{attribute 'qualified_only'}
VAR_GLOBAL
	bGetUp : BOOL := TRUE;
	bReady : BOOL;
END_VAR

(* stored: Version 1.1.0.1, ProductVersion 3.1.4024.12
   GVL GVL: Id {ac78c932-1368-4cfc-8235-67c46103f809} *)
